// Block: IPC_Com_Channel_LOG_MES

DATA_BLOCK IPC_Com_Channel_LOG_MES
VERSION : 0.1
   NON_RETAIN
   VAR
      RECEIVE : Struct
         ack : DInt;
         msg : IPC_Msg_Generico;
      END_STRUCT;
      SEND : Struct
         ack : DInt;
         msg : IPC_Msg_Log_MES;
      END_STRUCT;
   END_VAR

BEGIN
   // No initialization required
END_DATA_BLOCK
